PROGRAM uuidv7_g
VAR
	fbStartProcess : NT_StartProcess;
	step: INT;
END_VAR
VAR_OUTPUT
	bBuzy : BOOL;
	bDone : BOOL;
	bError : BOOL;
	UUID:STRING(36);
	ErrorID : UDINT;
END_VAR

CASE step OF
	1:
		UUID := '';
		fbStartProcess.START := FALSE;
		step := step + 1;
		
	2:
		fbStartProcess.START := TRUE;
		step := step + 1;
		
	3:
		IF fbStartProcess.BUSY OR fbStartProcess.ERR THEN
			step := step + 1;
		END_IF
		
	4:
		IF NOT fbStartProcess.BUSY AND NOT fbStartProcess.ERR THEN
			fbStartProcess.START := FALSE;
			step := step + 1;
		ELSIF fbStartProcess.ERR THEN
			fbStartProcess.START := FALSE;
			ErrorID := fbStartProcess.ERRID;
			step := step + 10000;
		END_IF
		
	5:
		IF Len(UUID) >= 36 THEN
			bDone := TRUE;
			step := 0;
		END_IF
END_CASE
	

bBuzy := step > 0 AND step < 10000;

bError := step > 10000;

IF bBuzy THEN
	bDone := FALSE;
END_IF

fbStartProcess(
		NETID := '',
		PATHSTR := 'C:\custom\uuidv7generator_ads\uuidv7generator_ads.exe',
		DIRNAME := 'C:\custom\uuidv7generator_ads',
		COMNDLINE := '127.0.0.1.1.1 851 uuidv7_g.UUID',
		TMOUT := T#1S
	);

METHOD Get
VAR_INPUT
END_VAR
step := 1;
END_METHOD

END_PROGRAM

(* stored: Version 1.1.0.1, ProductVersion 3.1.4026.13
   POU uuidv7_g: Id {02be623e-23c4-4422-bd23-1e6796f686de}, SpecialFunc None
   Method Get: Id {22afd9c5-56f5-40ef-af08-46603e18de3a} *)
